TYPE MassenstromSensor :
STRUCT
	ModbusAdresse:			BYTE := 12;
	Data: 					ARRAY[0..1] OF DWORD;	(*hier werden die abgefragen Register hineingeschrieben*)
	Startfeld_ModbusData: 	INT ; 
	
//------hier sind die Messwerte deklariert, die vom Massenstromsensor per Modbus erfragt werden	
	rMassenstrom: 					REAL; 					(*angegeben in kg/h*)
	rDruck: 						REAL;					(*in Bar*)
	rDichte: 						REAL;					(*kg/m³*)
	rTemp:							REAL;					(*angegeben in °C*)
	
	bFliessrichtung:				BOOL;					(*TRUE bei normaler Fließrichtung, FALSE bei Strömungsumkehrung*)

	
	
END_STRUCT
END_TYPE

(* stored: Version 1.1.0.1, ProductVersion 3.1.4019.2
   DUT MassenstromSensor: Id {a5e4a91b-adb7-4e42-b950-51204c2ef267} *)
